Omron CX-Programmer project NewProject (CX-Programmer 9.70)

# PLC NewPLC1: CP1L M

## Global symbols (name address type ; comment)
0.00 BOOL  ; SW1
0.01 BOOL  ; SW2
100.00 BOOL  ; LED1
100.01 BOOL  ; LED2
1.00 BOOL  ; LED1

## Program NewProgram1 (cyclic task 0)

### Section Section1

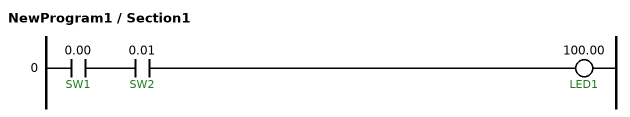
; rung 0
LD 0.00  ; SW1
AND 0.01  ; SW2
OUT 100.00  ; LED1

### Section END
; rung 0
END(001)